(* CODESYS project WagoLibGetLocationByIpAddress_v0.0.1.library
   Version: 0.0.1
   Author: Jesse Cox
   Title: WagoLibGetLocationByIpAddress
   Description: This library contains function blocks to get the hardware location using the gateway public IP address.
   Company: WAGO Corp. USA

Project tree, tasks and I/O mapping:
  libraries: SysProcess, 3.5.7.0 (System); Standard, * (System); WagoSysString, 1.6.0.0 (WAGO); SysTypes2 Interfaces, 3.5.4.0 (System); WagoAppFileDir, 1.6.1.1 (WAGO)
  data type LOCATION
  function block fbGetCurrentIpLocation [ST]: CurlGetCurrentLocation
*)

// LOCATION
TYPE LOCATION :
(*
{
    "ip": "71.237.213.64",
    "city": "Damascus",
    "region": "Oregon",
    "region_code": "OR",
    "country": "US",
    "country_name": "United States",
    "postal": "97089",
    "latitude": 45.4176,
    "longitude": -122.459,
    "timezone": "America/Los_Angeles",
    "asn": "AS7922",
    "org": "Comcast Cable Communications, LLC"
}
*)
STRUCT
	sPublicIpAddress	: STRING;
	sCity				: STRING;
	sState				: STRING;
	sStateCode			: STRING;
	sCountryCode		: STRING;
	sCountryName		: STRING;
	sPostalCode			: STRING;
	sLatitude			: STRING;
	sLongitude			: STRING;
END_STRUCT
END_TYPE

// fbGetCurrentIpLocation
FUNCTION_BLOCK fbGetCurrentIpLocation
VAR_IN_OUT
	xExecute			: BOOL;
END_VAR
VAR_INPUT
END_VAR
VAR_OUTPUT
	typCurrentLocation		: LOCATION;
END_VAR
VAR
	fbReadFile: FbReadWholeFile_cpt;
	oReadFileStatus: FbResult;
	xReadFileTrigger: BOOL;
	xReadFileError: BOOL;
	xReadFileBusy: BOOL;
	sReadFileName: STRING := '/root/location.json';
	aReadFileData: ARRAY[0..1000] OF BYTE;
	iReadFileSize: UDINT := 1000;
	iReadFileNumOfBytes: UDINT;
	xReadFileEndOfFileReached: BOOL;
	i: UDINT;
	
	sStringInProcess	: STRING;
	sProcessedStrings	: ARRAY[0..30] OF STRING;
	xIsCharacter: BOOL;
	ftCurlDoneTrig	: F_TRIG;
	rtFileIsDone	: R_TRIG;
	rtNotCharacter	: R_TRIG;
	iCharCount: INT;
END_VAR

IF xExecute THEN
	CurlGetCurrentLocation();
	xReadFileTrigger := TRUE;
END_IF

fbReadFile(
	oStatus=> oReadFileStatus, 
	xTrigger:= xReadFileTrigger, 
	xError=> xReadFileError, 
	xBusy=> xReadFileBusy, 
	sName:= sReadFileName, 
	pRxBuffer:= ADR(aReadFileData), 
	udiRxBufferSize:= iReadFileSize, 
	udiRxNBytes=> iReadFileNumOfBytes, 
	xEofReached=> xReadFileEndOfFileReached);
	
rtFileIsDone(CLK:= xReadFileEndOfFileReached);
iCharCount := 0; // reset the string count for processing
IF rtFileIsDone.Q THEN	
	FOR i := 0 TO iReadFileNumOfBytes DO
		IF 	((aReadFileData[i] >= 48) AND (aReadFileData[i] <= 57)) OR // characters 0-9
			((aReadFileData[i] >= 65) AND (aReadFileData[i] <= 90)) OR // characters A-Z
			((aReadFileData[i] >= 97) AND (aReadFileData[i] <= 122)) THEN // characters a-z
				xIsCharacter := TRUE;
		ELSIF 	(aReadFileData[i] = 34) OR // character "
				(aReadFileData[i] = 44) OR // character ,
				(aReadFileData[i] = 123) OR // character {
				(aReadFileData[i] = 125) THEN // character }
					xIsCharacter := FALSE;
		END_IF
	
		IF xIsCharacter THEN
			IF aReadFileData[i] = 32 THEN
				sStringInProcess := CONCAT(sStringInProcess, '_');
			ELSE
				sStringInProcess := CONCAT(sStringInProcess, ASCIIBYTE_TO_STRING(aReadFileData[i]));
			END_IF
				sProcessedStrings[iCharCount] := sStringInProcess;
		END_IF
			
		rtNotCharacter(CLK := NOT xIsCharacter);
		IF rtNotCharacter.Q THEN
			sStringInProcess := '';
			iCharCount := iCharCount + 1;
		END_IF
	END_FOR

	FOR i := 0 TO iCharCount DO
		IF sProcessedStrings[i] = 'city' THEN
			typCurrentLocation.sCity := sProcessedStrings[i + 1];	
		ELSIF sProcessedStrings[i] = 'region' THEN
			typCurrentLocation.sState := sProcessedStrings[i + 1];
		ELSIF sProcessedStrings[i] = 'regionName' THEN
			typCurrentLocation.sStateCode := sProcessedStrings[i + 1];
		ELSIF sProcessedStrings[i] = 'country' THEN
			typCurrentLocation.sCountryCode := sProcessedStrings[i + 1];
		ELSIF sProcessedStrings[i] = 'countryCode' THEN
			typCurrentLocation.sCountryName := sProcessedStrings[i + 1];
		ELSIF sProcessedStrings[i] = 'lat' THEN
			typCurrentLocation.sLatitude := sProcessedStrings[i + 1];
		ELSIF sProcessedStrings[i] = 'lon' THEN
			typCurrentLocation.sLongitude := sProcessedStrings[i + 1];
		ELSIF sProcessedStrings[i] = 'zip' THEN
			typCurrentLocation.sPostalCode := sProcessedStrings[i + 1];
		ELSIF sProcessedStrings[i] = 'query' THEN
			typCurrentLocation.sPublicIpAddress := sProcessedStrings[i + 1];
		END_IF
	END_FOR
	xExecute := FALSE;
END_IF

METHOD CurlGetCurrentLocation : STRING
VAR_INPUT
	//sApiKey		: STRING;
	//sApiState	: STRING;
	//sApiCity	: STRING;
END_VAR
VAR 
	sUprString	: STRING(255) := 'curl --insecure --output /root/location.json -X GET http://ip-api.com/json';	// base string to query location service
	diFileStatus: DINT;
	sQueryBashScript: STRING;
	sBashResponse: STRING;
	ptBashRslt: POINTER TO RTS_IEC_RESULT;
END_VAR
diFileStatus := SysProcessExecuteCommand2(pszCommand:= sUprString, pszStdOut:= sBashResponse, udiStdOutLen:= LEN(sUprString), pResult:= ptBashRslt);
//curl --insecure --output /root/weather.json -X GET http://api.wunderground.com/api/1ad24b0986c7e326/conditions/q/OR/Portland.json
END_METHOD

END_FUNCTION_BLOCK
